FUNCTION BYTES_TO_WORD
  (* Standard: 61499-1 *)
  (* Version 1.0, 2024-02-22, franz *)
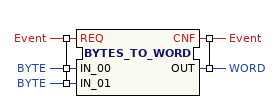
  EVENT_INPUT
    REQ WITH IN_00, IN_01; (* Normal Execution Request *)
  END_EVENT
  EVENT_OUTPUT
    CNF WITH OUT; (* Execution Confirmation *)
  END_EVENT
  VAR_INPUT
    IN_00 : BYTE; (* BYTE 00 *)
    IN_01 : BYTE; (* BYTE 01 *)
  END_VAR
  VAR_OUTPUT
    OUT : WORD; (* WORD Output *)
  END_VAR
  BODY IN ST:
FUNCTION BYTES_TO_WORD

VAR_INPUT
	IN_00 : BYTE;    // BYTE 00
	IN_01 : BYTE;    // BYTE 01
END_VAR

VAR_OUTPUT
	OUT : WORD;    // WORD Output
END_VAR

(* this Function combines the 2 BYTES to a word *)
OUT := SHL(IN_01, SHFT_BYTE_01)
	OR SHL(IN_00, SHFT_BYTE_00);

END_FUNCTION
  END_BODY
END_FUNCTION
